{attribute 'qualified_only'}
{attribute 'strict'}
TYPE E_AteqCallerState :
(
	INIT,		// Runs FB_init for al instances
	CONTROL		// Maps Io and Controls in RT
);
END_TYPE

(* stored: Version 1.1.0.1, ProductVersion 3.1.4024.15
   DUT E_AteqCallerState: Id {09bb713a-d2d4-40c1-bad9-0b2a11fda991} *)
